{attribute 'GeneratedUsingTerminal: EL6201-0000-0017'}
{attribute addProperty BoxType "EL6201-0000-0017"}
{attribute addProperty Id "Slave_1_OutputsAT %Q*Slave_1_Outputs_820A30FD8Slave_2_OutputsAT %Q*Slave_2_Outputs_EF052D198Slave_3_OutputsAT %Q*Slave_3_Outputs_37BF2D288Slave_4_OutputsAT %Q*Slave_4_Outputs_351B16D18Slave_5_OutputsAT %Q*Slave_5_Outputs_EDA116E08Slave_6_OutputsAT %Q*Slave_6_Outputs_80AE0B048Slave_7_OutputsAT %Q*Slave_7_Outputs_58140B358Slave_8_OutputsAT %Q*Slave_8_Outputs_85E67CF68Slave_9_OutputsAT %Q*Slave_9_Outputs_5D5C7CC78Slave_10_OutputsAT %Q*Slave_10_Outputs_0FEEBBCA8Slave_11_OutputsAT %Q*Slave_11_Outputs_DC7C3E208Slave_12_OutputsAT %Q*Slave_12_Outputs_AC0AADA98Slave_13_OutputsAT %Q*Slave_13_Outputs_7F9828438Slave_14_OutputsAT %Q*Slave_14_Outputs_4CE78ABB8Slave_15_OutputsAT %Q*Slave_15_Outputs_9F750F518Slave_16_OutputsAT %Q*Slave_16_Outputs_EF039CD88Slave_17_OutputsAT %Q*Slave_17_Outputs_3C9119328Slave_18_OutputsAT %Q*Slave_18_Outputs_89FCD9288Slave_19_OutputsAT %Q*Slave_19_Outputs_5A6E5CC28Slave_20_OutputsAT %Q*Slave_20_Outputs_99C92F2D8Slave_21_OutputsAT %Q*Slave_21_Outputs_4A5BAAC78Slave_22_OutputsAT %Q*Slave_22_Outputs_3A2D394E8Slave_23_OutputsAT %Q*Slave_23_Outputs_E9BFBCA48Slave_24_OutputsAT %Q*Slave_24_Outputs_DAC01E5C8Slave_25_OutputsAT %Q*Slave_25_Outputs_09529BB68Slave_26_OutputsAT %Q*Slave_26_Outputs_7924083F8Slave_27_OutputsAT %Q*Slave_27_Outputs_AAB68DD58Slave_28_OutputsAT %Q*Slave_28_Outputs_1FDB4DCF8Slave_29_OutputsAT %Q*Slave_29_Outputs_CC49C8258Slave_30_OutputsAT %Q*Slave_30_Outputs_1794A81D8Slave_31_OutputsAT %Q*Slave_31_Outputs_C4062DF78"}
{attribute addProperty CRC "369323545"}
{attribute addProperty Size "248"}
TYPE ASI_Outputs_Device_16036E19 EXTENDS OutputBase_10CEE7DE :
STRUCT
	{attribute addProperty Name "Slave_1_Outputs"}
	Slave_1_Outputs AT %Q* : Slave_1_Outputs_820A30FD;
	{attribute addProperty Name "Slave_2_Outputs"}
	Slave_2_Outputs AT %Q* : Slave_2_Outputs_EF052D19;
	{attribute addProperty Name "Slave_3_Outputs"}
	Slave_3_Outputs AT %Q* : Slave_3_Outputs_37BF2D28;
	{attribute addProperty Name "Slave_4_Outputs"}
	Slave_4_Outputs AT %Q* : Slave_4_Outputs_351B16D1;
	{attribute addProperty Name "Slave_5_Outputs"}
	Slave_5_Outputs AT %Q* : Slave_5_Outputs_EDA116E0;
	{attribute addProperty Name "Slave_6_Outputs"}
	Slave_6_Outputs AT %Q* : Slave_6_Outputs_80AE0B04;
	{attribute addProperty Name "Slave_7_Outputs"}
	Slave_7_Outputs AT %Q* : Slave_7_Outputs_58140B35;
	{attribute addProperty Name "Slave_8_Outputs"}
	Slave_8_Outputs AT %Q* : Slave_8_Outputs_85E67CF6;
	{attribute addProperty Name "Slave_9_Outputs"}
	Slave_9_Outputs AT %Q* : Slave_9_Outputs_5D5C7CC7;
	{attribute addProperty Name "Slave_10_Outputs"}
	Slave_10_Outputs AT %Q* : Slave_10_Outputs_0FEEBBCA;
	{attribute addProperty Name "Slave_11_Outputs"}
	Slave_11_Outputs AT %Q* : Slave_11_Outputs_DC7C3E20;
	{attribute addProperty Name "Slave_12_Outputs"}
	Slave_12_Outputs AT %Q* : Slave_12_Outputs_AC0AADA9;
	{attribute addProperty Name "Slave_13_Outputs"}
	Slave_13_Outputs AT %Q* : Slave_13_Outputs_7F982843;
	{attribute addProperty Name "Slave_14_Outputs"}
	Slave_14_Outputs AT %Q* : Slave_14_Outputs_4CE78ABB;
	{attribute addProperty Name "Slave_15_Outputs"}
	Slave_15_Outputs AT %Q* : Slave_15_Outputs_9F750F51;
	{attribute addProperty Name "Slave_16_Outputs"}
	Slave_16_Outputs AT %Q* : Slave_16_Outputs_EF039CD8;
	{attribute addProperty Name "Slave_17_Outputs"}
	Slave_17_Outputs AT %Q* : Slave_17_Outputs_3C911932;
	{attribute addProperty Name "Slave_18_Outputs"}
	Slave_18_Outputs AT %Q* : Slave_18_Outputs_89FCD928;
	{attribute addProperty Name "Slave_19_Outputs"}
	Slave_19_Outputs AT %Q* : Slave_19_Outputs_5A6E5CC2;
	{attribute addProperty Name "Slave_20_Outputs"}
	Slave_20_Outputs AT %Q* : Slave_20_Outputs_99C92F2D;
	{attribute addProperty Name "Slave_21_Outputs"}
	Slave_21_Outputs AT %Q* : Slave_21_Outputs_4A5BAAC7;
	{attribute addProperty Name "Slave_22_Outputs"}
	Slave_22_Outputs AT %Q* : Slave_22_Outputs_3A2D394E;
	{attribute addProperty Name "Slave_23_Outputs"}
	Slave_23_Outputs AT %Q* : Slave_23_Outputs_E9BFBCA4;
	{attribute addProperty Name "Slave_24_Outputs"}
	Slave_24_Outputs AT %Q* : Slave_24_Outputs_DAC01E5C;
	{attribute addProperty Name "Slave_25_Outputs"}
	Slave_25_Outputs AT %Q* : Slave_25_Outputs_09529BB6;
	{attribute addProperty Name "Slave_26_Outputs"}
	Slave_26_Outputs AT %Q* : Slave_26_Outputs_7924083F;
	{attribute addProperty Name "Slave_27_Outputs"}
	Slave_27_Outputs AT %Q* : Slave_27_Outputs_AAB68DD5;
	{attribute addProperty Name "Slave_28_Outputs"}
	Slave_28_Outputs AT %Q* : Slave_28_Outputs_1FDB4DCF;
	{attribute addProperty Name "Slave_29_Outputs"}
	Slave_29_Outputs AT %Q* : Slave_29_Outputs_CC49C825;
	{attribute addProperty Name "Slave_30_Outputs"}
	Slave_30_Outputs AT %Q* : Slave_30_Outputs_1794A81D;
	{attribute addProperty Name "Slave_31_Outputs"}
	Slave_31_Outputs AT %Q* : Slave_31_Outputs_C4062DF7;
END_STRUCT
END_TYPE

(* stored: Version 1.2.0.0, ProductVersion 3.1.4024.9
   DUT ASI_Outputs_Device_16036E19: Id {21401d8f-5037-406a-abc4-99417d1ff7d5} *)
